FUNCTION_BLOCK XSPACE (* A spacer object with center and edge labels *)
  (* Standard: 61499-1; Function: HMI; Type: Spacer *)
  (* Version 0.0, 2001-03-08, JHC, Rockwell Automation, First XML version. *)
  (* Compiler header: package fb.rt.hmi; import java.awt.*; *)
  (* Compiler Java IBM VisualAge 3.0 *)
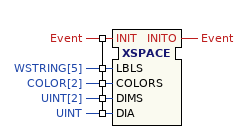
  EVENT_INPUT
    INIT WITH LBLS, COLORS, DIMS, DIA; (* Initialize *)
  END_EVENT
  EVENT_OUTPUT
    INITO; (* Initialization Confirm *)
  END_EVENT
  VAR_INPUT
    LBLS : ARRAY [0..4] OF WSTRING; (* Labels:{Left,Top,Right,Bottom,Center} *)
    COLORS : ARRAY [0..1] OF COLOR := [black,white]; (* {Foreground,Background} *)
    DIMS : ARRAY [0..1] OF UINT := [3,3]; (* {Width,Height}in Diameters *)
    DIA : UINT := 25; (* Diameter dimension *)
  END_VAR
END_FUNCTION_BLOCK
